(* PLC project Untitled1, Beckhoff Automation GmbH TwinCAT PLC Control 3.5.20.40 *)
(* stored: creationDateTime 2025-05-07T14:52:09.5185914, modificationDateTime 2025-05-07T14:52:09.5215848 *)

PROGRAM MAIN
VAR
	
bInit : BOOL := TRUE; 
    bSend : BOOL := TRUE; 

    fbMsg : FB_TcMessage; 
	
	test : BOOL;

END_VAR

                  IF bInit THEN
    bInit := FALSE; 
    fbMsg.CreateEx(TC_EVENTS.EventTest.Help, 0); 
	fbMsg.CreateEx(TC_EVENTS.EventTest.Help2, 0);
	//fbMsg.CreateEx(TC_EVENTS.EventTest.Help3, 0);
END_IF

IF bSend THEN 
    bSend := FALSE; 
    fbMsg.Send(0); 
END_IF
                
END_PROGRAM

CONFIGURATION Application
  RESOURCE Untitled1 ON PLC
    TASK PlcTask(INTERVAL := T#0ms, PRIORITY := 20);
    PROGRAM MAIN WITH PlcTask : MAIN;
  END_RESOURCE
END_CONFIGURATION
